TYPE ST115_Pnp_e : ST110_Pnp_e;
END_TYPE

(* stored: Version 1.1.0.1, ProductVersion 3.1.4024.6
   EnumerationTextList ST115_Pnp_e: Id {9006f64b-f8ec-4be8-a84e-61da86b4eb29} *)
